TYPE "ValveMachine_DataIn"
VERSION : 0.1
// Block: ValveMachine_DataIn
   STRUCT
      PB : ValveMachine_PB;
      Rest_Ls : Array[1..8] of Bool;
      Work_Ls : Array[1..8] of Bool;
   END_STRUCT;

END_TYPE
